(* Schneider Machine Expert - Basic project Questao4.1_FelipeV1_20241016, file version 2.9.0.0 *)
(* ProjectInformations: Name=Novo projeto *)

HARDWARE
  Cpu 0: TM221M16R/G
  EthernetConfiguration: NetworkName=M221, IpAllocationMode=FixedAddress, IpAddress=0.0.0.0, SubnetMask=0.0.0.0
  SerialLineConfiguration: Baud=Baud19200, Parity=ParityEven, DataBits=DataBits8, StopBits=StopBits1, PhysicalMedium=PhysicalMediumRs485, TransmissionMode=TransmissionModeModbusRtu, SlaveId=1, Addressing=SlaveAddressing
  MastTask: UsePeriodScanMode=false, PeriodScan=100
  FastTask: Period=255
  CpuBehavior: StartingMode=StartAsPreviousState, AutoSaveRamOnEeprom=true, WatchdogPeriod=250

SYMBOLS  (address, symbol, comment, settings)
  %M5       TRAN_1_TO_2
  %M6       TRAN_2_TO_3
  %M7       TRAN_3_TO_4
  %M8       TRAN_4_TO_1
  %M10      SINAL_VERD_VIA_1
  %M11      SINAL_AMAR_VIA_1
  %M12      SINAL_VERM_VIA_1
  %M20      SINAL_VERD_VIA_2
  %M21      SINAL_AMAR_VIA_2
  %M22      SINAL_VERM_VIA_2
  %X1       TRAN_1
  %X2       TRAN_2
  %X3       TRAN_3
  %X4       TRAN_4
  %TM0      FT_1_TO_2  [Preset=27, Base=OneSecond]
  %TM1      FT_2_TO_3  [Preset=3, Base=OneSecond]
  %TM2      FT_3_TO_4  [Preset=27, Base=OneSecond]
  %TM3      FT_4_TO_1  [Preset=3, Base=OneSecond]
  %Q0.1     SAIDA_SINAL_VERD_VIA_1
  %Q0.2     SAIDA_SINAL_AMAR_VIA_1
  %Q0.3     SAIDA_SINAL_VERM_VIA_1
  %Q0.4     SAIDA_SINAL_VERD_VIA_2
  %Q0.5     SAIDA_SINAL_AMAR_VIA_2
  %Q0.6     SAIDA_SINAL_VERM_VIA_2

GRAFCET Grafcet POU
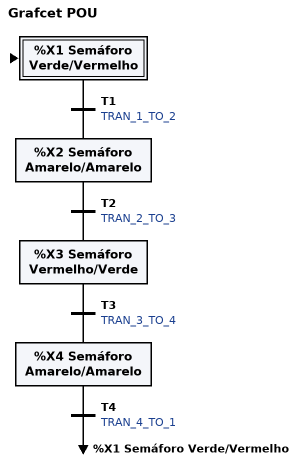
  INITIAL_STEP %X1  (* Semáforo Verde/Vermelho *)
  STEP %X2  (* Semáforo Amarelo/Amarelo *)
  STEP %X3  (* Semáforo Vermelho/Verde *)
  STEP %X4  (* Semáforo Amarelo/Amarelo *)
  TRANSITION T1 FROM %X1 TO %X2 := TRAN_1_TO_2;
  TRANSITION T2 FROM %X2 TO %X3 := TRAN_2_TO_3;
  TRANSITION T3 FROM %X3 TO %X4 := TRAN_3_TO_4;
  TRANSITION T4 FROM %X4 TO %X1 := TRAN_4_TO_1;

TRANSITION T1 (%X1 -> %X2) 
  (* SectionNumber=0 *)

// Rung 0: TRAN E1 TO E2
  LD %M5                  (* TRAN_1_TO_2 *)
  ENDT
  // as ST:
  //   TRANSITION := TRAN_1_TO_2;

TRANSITION T2 (%X2 -> %X3) 
  (* SectionNumber=0 *)

// Rung 1: TRAN E2 TO E3
  LD %M6                  (* TRAN_2_TO_3 *)
  ENDT
  // as ST:
  //   TRANSITION := TRAN_2_TO_3;

TRANSITION T3 (%X3 -> %X4) 
  (* SectionNumber=0 *)

// Rung 2: TRAN E3 TO E4
  LD %M7                  (* TRAN_3_TO_4 *)
  ENDT
  // as ST:
  //   TRANSITION := TRAN_3_TO_4;

TRANSITION T4 (%X4 -> %X1) 
  (* SectionNumber=0 *)

// Rung 3: TRAN E4 TO E1
  LD %M8                  (* TRAN_4_TO_1 *)
  ENDT
  // as ST:
  //   TRANSITION := TRAN_4_TO_1;

POU Lógica
  (* SectionNumber=5 *)

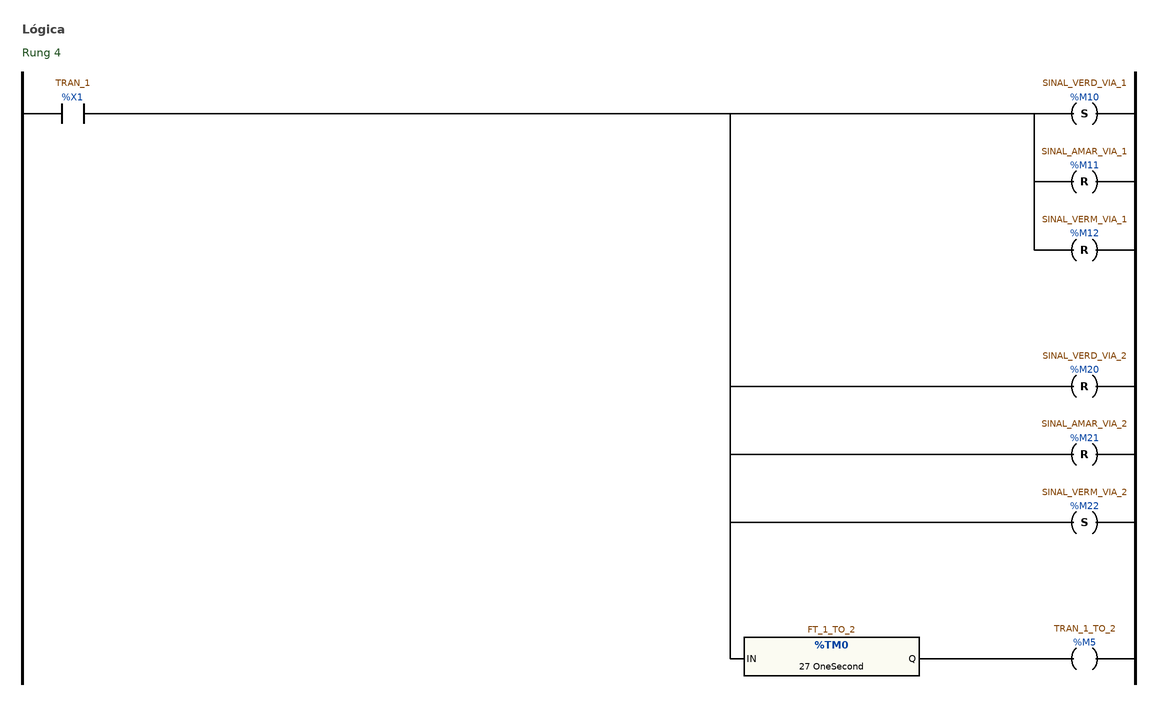

// Rung 4
  LD 1
  MULTIFB
  LD 1
  AND %X1                 (* TRAN_1 *)
  ST %MW2009:X0
  LD %MW2009:X0
  S %M10                  (* SINAL_VERD_VIA_1 *)
  R %M11                  (* SINAL_AMAR_VIA_1 *)
  R %M12                  (* SINAL_VERM_VIA_1 *)
  R %M20                  (* SINAL_VERD_VIA_2 *)
  R %M21                  (* SINAL_AMAR_VIA_2 *)
  S %M22                  (* SINAL_VERM_VIA_2 *)
  BLK %TM0                (* FT_1_TO_2 *)
  LD %MW2009:X0
  IN
  OUT_BLK
  LD Q
  ST %M5                  (* TRAN_1_TO_2 *)
  END_BLK
  MULTIFB
  // as ST:
  //   IF TRAN_1 THEN SINAL_VERD_VIA_1 := TRUE; END_IF;
  //   IF TRAN_1 THEN SINAL_AMAR_VIA_1 := FALSE; END_IF;
  //   IF TRAN_1 THEN SINAL_VERM_VIA_1 := FALSE; END_IF;
  //   IF TRAN_1 THEN SINAL_VERD_VIA_2 := FALSE; END_IF;
  //   IF TRAN_1 THEN SINAL_AMAR_VIA_2 := FALSE; END_IF;
  //   IF TRAN_1 THEN SINAL_VERM_VIA_2 := TRUE; END_IF;
  //   FT_1_TO_2(IN := TRAN_1);
  //   TRAN_1_TO_2 := FT_1_TO_2.Q;

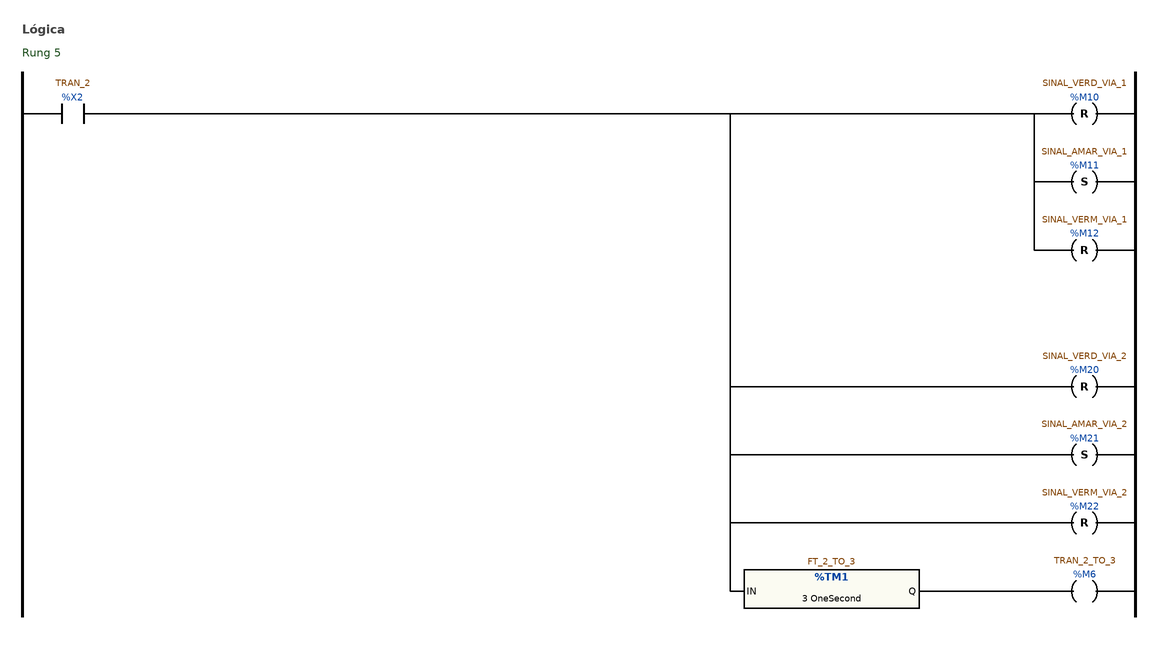

// Rung 5
  LD 1
  MULTIFB
  LD 1
  AND %X2                 (* TRAN_2 *)
  ST %MW2009:X0
  LD %MW2009:X0
  R %M10                  (* SINAL_VERD_VIA_1 *)
  S %M11                  (* SINAL_AMAR_VIA_1 *)
  R %M12                  (* SINAL_VERM_VIA_1 *)
  R %M20                  (* SINAL_VERD_VIA_2 *)
  S %M21                  (* SINAL_AMAR_VIA_2 *)
  R %M22                  (* SINAL_VERM_VIA_2 *)
  BLK %TM1                (* FT_2_TO_3 *)
  LD %MW2009:X0
  IN
  OUT_BLK
  LD Q
  ST %M6                  (* TRAN_2_TO_3 *)
  END_BLK
  MULTIFB
  // as ST:
  //   IF TRAN_2 THEN SINAL_VERD_VIA_1 := FALSE; END_IF;
  //   IF TRAN_2 THEN SINAL_AMAR_VIA_1 := TRUE; END_IF;
  //   IF TRAN_2 THEN SINAL_VERM_VIA_1 := FALSE; END_IF;
  //   IF TRAN_2 THEN SINAL_VERD_VIA_2 := FALSE; END_IF;
  //   IF TRAN_2 THEN SINAL_AMAR_VIA_2 := TRUE; END_IF;
  //   IF TRAN_2 THEN SINAL_VERM_VIA_2 := FALSE; END_IF;
  //   FT_2_TO_3(IN := TRAN_2);
  //   TRAN_2_TO_3 := FT_2_TO_3.Q;

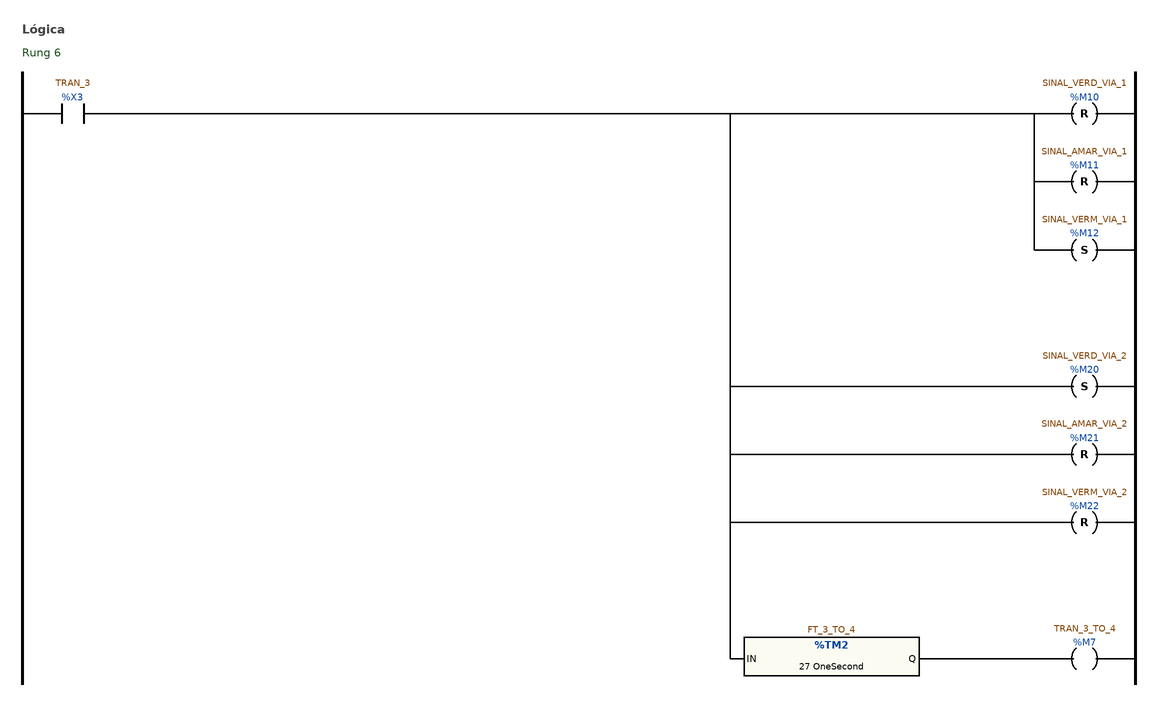

// Rung 6
  LD 1
  MULTIFB
  LD 1
  AND %X3                 (* TRAN_3 *)
  ST %MW2009:X0
  LD %MW2009:X0
  R %M10                  (* SINAL_VERD_VIA_1 *)
  R %M11                  (* SINAL_AMAR_VIA_1 *)
  S %M12                  (* SINAL_VERM_VIA_1 *)
  S %M20                  (* SINAL_VERD_VIA_2 *)
  R %M21                  (* SINAL_AMAR_VIA_2 *)
  R %M22                  (* SINAL_VERM_VIA_2 *)
  BLK %TM2                (* FT_3_TO_4 *)
  LD %MW2009:X0
  IN
  OUT_BLK
  LD Q
  ST %M7                  (* TRAN_3_TO_4 *)
  END_BLK
  MULTIFB
  // as ST:
  //   IF TRAN_3 THEN SINAL_VERD_VIA_1 := FALSE; END_IF;
  //   IF TRAN_3 THEN SINAL_AMAR_VIA_1 := FALSE; END_IF;
  //   IF TRAN_3 THEN SINAL_VERM_VIA_1 := TRUE; END_IF;
  //   IF TRAN_3 THEN SINAL_VERD_VIA_2 := TRUE; END_IF;
  //   IF TRAN_3 THEN SINAL_AMAR_VIA_2 := FALSE; END_IF;
  //   IF TRAN_3 THEN SINAL_VERM_VIA_2 := FALSE; END_IF;
  //   FT_3_TO_4(IN := TRAN_3);
  //   TRAN_3_TO_4 := FT_3_TO_4.Q;

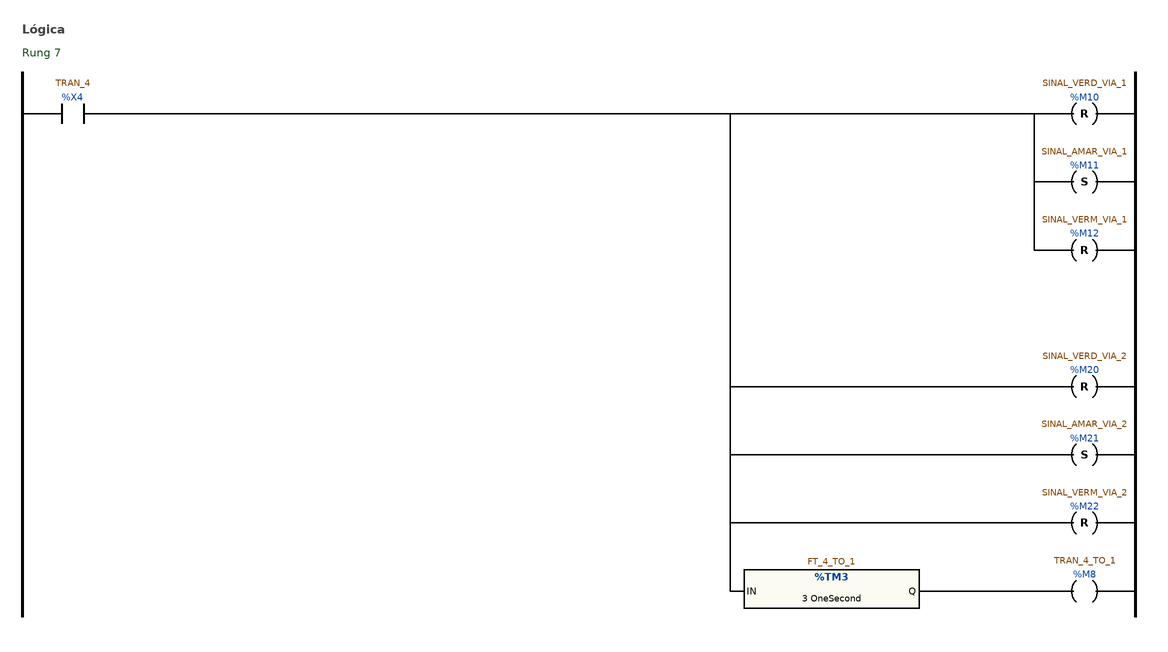

// Rung 7
  LD 1
  MULTIFB
  LD 1
  AND %X4                 (* TRAN_4 *)
  ST %MW2009:X0
  LD %MW2009:X0
  R %M10                  (* SINAL_VERD_VIA_1 *)
  S %M11                  (* SINAL_AMAR_VIA_1 *)
  R %M12                  (* SINAL_VERM_VIA_1 *)
  R %M20                  (* SINAL_VERD_VIA_2 *)
  S %M21                  (* SINAL_AMAR_VIA_2 *)
  R %M22                  (* SINAL_VERM_VIA_2 *)
  BLK %TM3                (* FT_4_TO_1 *)
  LD %MW2009:X0
  IN
  OUT_BLK
  LD Q
  ST %M8                  (* TRAN_4_TO_1 *)
  END_BLK
  MULTIFB
  // as ST:
  //   IF TRAN_4 THEN SINAL_VERD_VIA_1 := FALSE; END_IF;
  //   IF TRAN_4 THEN SINAL_AMAR_VIA_1 := TRUE; END_IF;
  //   IF TRAN_4 THEN SINAL_VERM_VIA_1 := FALSE; END_IF;
  //   IF TRAN_4 THEN SINAL_VERD_VIA_2 := FALSE; END_IF;
  //   IF TRAN_4 THEN SINAL_AMAR_VIA_2 := TRUE; END_IF;
  //   IF TRAN_4 THEN SINAL_VERM_VIA_2 := FALSE; END_IF;
  //   FT_4_TO_1(IN := TRAN_4);
  //   TRAN_4_TO_1 := FT_4_TO_1.Q;

POU Saída
  (* SectionNumber=0 *)

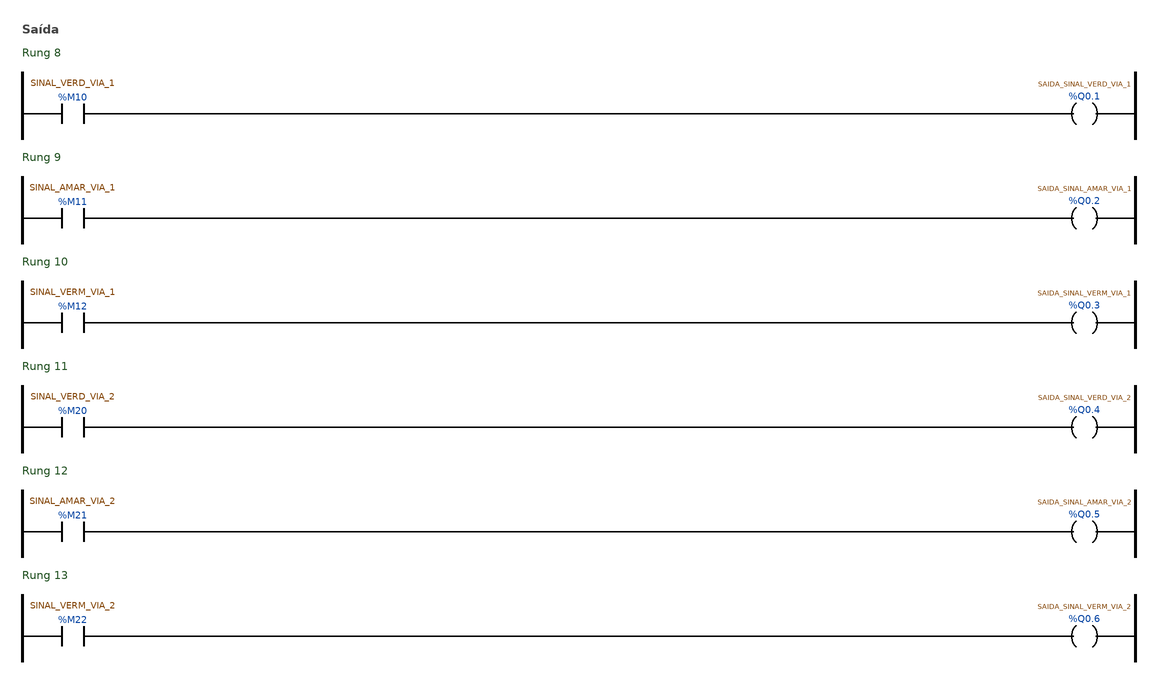

// Rung 8
  LD %M10                 (* SINAL_VERD_VIA_1 *)
  ST %Q0.1                (* SAIDA_SINAL_VERD_VIA_1 *)
  // as ST:
  //   SAIDA_SINAL_VERD_VIA_1 := SINAL_VERD_VIA_1;

// Rung 9
  LD %M11                 (* SINAL_AMAR_VIA_1 *)
  ST %Q0.2                (* SAIDA_SINAL_AMAR_VIA_1 *)
  // as ST:
  //   SAIDA_SINAL_AMAR_VIA_1 := SINAL_AMAR_VIA_1;

// Rung 10
  LD %M12                 (* SINAL_VERM_VIA_1 *)
  ST %Q0.3                (* SAIDA_SINAL_VERM_VIA_1 *)
  // as ST:
  //   SAIDA_SINAL_VERM_VIA_1 := SINAL_VERM_VIA_1;

// Rung 11
  LD %M20                 (* SINAL_VERD_VIA_2 *)
  ST %Q0.4                (* SAIDA_SINAL_VERD_VIA_2 *)
  // as ST:
  //   SAIDA_SINAL_VERD_VIA_2 := SINAL_VERD_VIA_2;

// Rung 12
  LD %M21                 (* SINAL_AMAR_VIA_2 *)
  ST %Q0.5                (* SAIDA_SINAL_AMAR_VIA_2 *)
  // as ST:
  //   SAIDA_SINAL_AMAR_VIA_2 := SINAL_AMAR_VIA_2;

// Rung 13
  LD %M22                 (* SINAL_VERM_VIA_2 *)
  ST %Q0.6                (* SAIDA_SINAL_VERM_VIA_2 *)
  // as ST:
  //   SAIDA_SINAL_VERM_VIA_2 := SINAL_VERM_VIA_2;
